// TIA Portal project "Automação_Grupo_2_V0.2" (V16)

(* hardware
DEVICE "S7-1200 station_1"  S7-1200 Station
   slot 0: "Rack_0"  S7-1200 Rack  Rack  V1.0
   slot 1: "PLC_1"  CPU 1211C AC/DC/Rly  6ES7 211-1BE40-0XB0  V4.4
   slot 3: "DI 4x24VDC_1"  DI4 signal board (200 kHz)  6ES7 221-3BD30-0XB0  V1.0
*)

// ===== PLC "PLC_1"  CPU 1211C AC/DC/Rly =====

VAR_GLOBAL   // PLC tag table "Default tag table"
   "Start(NO)" AT %I0.0 : Bool;
   "Stop(NC)" AT %I0.1 : Bool;
   "Reset(NO)" AT %I0.2 : Bool;
   "Emergência(NO)" AT %I0.3 : Bool;
   "Sensor Final (NO) AV PART1" AT %I0.4 : Bool;
   "Cilindro Alimentador Avanço" AT %I0.5 : Bool;
   "Peça no Alimentador" AT %I1.0 : Bool;
   "Sensor Fase 1 (NO)" AT %I1.1 : Bool;
   "Sensor Fase 2 (NO)" AT %I1.2 : Bool;
   "Sensor Fase 3 (NC)" AT %I1.3 : Bool;
   "Ordem Direita" AT %Q0.0 : Bool;
   "Ordem Esquerda" AT %Q0.1 : Bool;
   "Avanço Cilindro de Alimentação" AT %Q0.2 : Bool;
   "Seletor de Peças do Conveyor" AT %Q0.3 : Bool;
   "E_Verificação" AT %M0.1 : Bool;
   "E_2" AT %M0.2 : Bool;
   "E_3" AT %M0.3 : Bool;
   "E_4" AT %M0.4 : Bool;
   "E_5" AT %M0.5 : Bool;
   "E_6" AT %M0.6 : Bool;
   "E_7" AT %M0.7 : Bool;
   "E_8" AT %M1.0 : Bool;
   "E_9" AT %M1.1 : Bool;
   "E_10" AT %M1.2 : Bool;
   "T1_STATUS" AT %M1.3 : Bool;
END_VAR

// folder: System blocks/Program resources

DATA_BLOCK "T1"   // DB1
{ S7_Optimized_Access := 'TRUE' }
AUTHOR : Simatic
FAMILY : IEC
NAME : IEC_TMR
VERSION : 1.0
// stored: InstanceOfName IEC_TIMER
"IEC_TIMER"
BEGIN
END_DATA_BLOCK

DATA_BLOCK "Temporizador 01"   // DB2
{ S7_Optimized_Access := 'TRUE' }
AUTHOR : Simatic
FAMILY : IEC
NAME : IEC_TMR
VERSION : 1.0
// stored: InstanceOfName IEC_TIMER
"IEC_TIMER"
BEGIN
END_DATA_BLOCK

DATA_BLOCK "Cooldown para Motor"   // DB3
{ S7_Optimized_Access := 'TRUE' }
AUTHOR : Simatic
FAMILY : IEC
NAME : IEC_TMR
VERSION : 1.0
// stored: InstanceOfName IEC_TIMER
"IEC_TIMER"
BEGIN
END_DATA_BLOCK

DATA_BLOCK "COoldown para Desligar Esquerda"   // DB4
{ S7_Optimized_Access := 'TRUE' }
AUTHOR : Simatic
FAMILY : IEC
NAME : IEC_TMR
VERSION : 1.0
// stored: InstanceOfName IEC_TIMER
"IEC_TIMER"
BEGIN
END_DATA_BLOCK

DATA_BLOCK "Temporizador para Direita"   // DB5
{ S7_Optimized_Access := 'TRUE' }
AUTHOR : Simatic
FAMILY : IEC
NAME : IEC_TMR
VERSION : 1.0
// stored: InstanceOfName IEC_TIMER
"IEC_TIMER"
BEGIN
END_DATA_BLOCK

DATA_BLOCK "XTempo do Seletor"   // DB6
{ S7_Optimized_Access := 'TRUE' }
AUTHOR : Simatic
FAMILY : IEC
NAME : IEC_TMR
VERSION : 1.0
// stored: InstanceOfName IEC_TIMER
"IEC_TIMER"
BEGIN
END_DATA_BLOCK

DATA_BLOCK "Cooldown Estação 2"   // DB7
{ S7_Optimized_Access := 'TRUE' }
AUTHOR : Simatic
FAMILY : IEC
NAME : IEC_TMR
VERSION : 1.0
// stored: InstanceOfName IEC_TIMER
"IEC_TIMER"
BEGIN
END_DATA_BLOCK

DATA_BLOCK "5 Segundos 2a Estação"   // DB8
{ S7_Optimized_Access := 'TRUE' }
AUTHOR : Simatic
FAMILY : IEC
NAME : IEC_TMR
VERSION : 1.0
// stored: InstanceOfName IEC_TIMER
"IEC_TIMER"
BEGIN
END_DATA_BLOCK

DATA_BLOCK "Cooldown para fechar o Seletor"   // DB9
{ S7_Optimized_Access := 'TRUE' }
AUTHOR : Simatic
FAMILY : IEC
NAME : IEC_TMR
VERSION : 1.0
// stored: InstanceOfName IEC_TIMER
"IEC_TIMER"
BEGIN
END_DATA_BLOCK

DATA_BLOCK "Cooldown para Terminar Processo"   // DB10
{ S7_Optimized_Access := 'TRUE' }
AUTHOR : Simatic
FAMILY : IEC
NAME : IEC_TMR
VERSION : 1.0
// stored: InstanceOfName IEC_TIMER
"IEC_TIMER"
BEGIN
END_DATA_BLOCK

DATA_BLOCK "Cooldown para DEsligar mOtor 3a Estação"   // DB11
{ S7_Optimized_Access := 'TRUE' }
AUTHOR : Simatic
FAMILY : IEC
NAME : IEC_TMR
VERSION : 1.0
// stored: InstanceOfName IEC_TIMER
"IEC_TIMER"
BEGIN
END_DATA_BLOCK

DATA_BLOCK "condição de entrada e8+e9"   // DB12
{ S7_Optimized_Access := 'TRUE' }
AUTHOR : Simatic
FAMILY : IEC
NAME : IEC_TMR
VERSION : 1.0
// stored: InstanceOfName IEC_TIMER
"IEC_TIMER"
BEGIN
END_DATA_BLOCK

DATA_BLOCK "contador de peças"   // DB13
{ S7_Optimized_Access := 'TRUE' }
AUTHOR : Simatic
FAMILY : IEC
NAME : CNTR
VERSION : 1.0
// stored: InstanceOfName IEC_COUNTER
"IEC_COUNTER"
BEGIN
END_DATA_BLOCK

DATA_BLOCK "cooldown para mandar pecas novamente"   // DB14
{ S7_Optimized_Access := 'TRUE' }
AUTHOR : Simatic
FAMILY : IEC
NAME : IEC_TMR
VERSION : 1.0
// stored: InstanceOfName IEC_TIMER
"IEC_TIMER"
BEGIN
END_DATA_BLOCK

DATA_BLOCK "cooldown final"   // DB15
{ S7_Optimized_Access := 'TRUE' }
AUTHOR : Simatic
FAMILY : IEC
NAME : IEC_TMR
VERSION : 1.0
// stored: InstanceOfName IEC_TIMER
"IEC_TIMER"
BEGIN
END_DATA_BLOCK

DATA_BLOCK "cooldown para peça retirada"   // DB16
{ S7_Optimized_Access := 'TRUE' }
AUTHOR : Simatic
FAMILY : IEC
NAME : IEC_TMR
VERSION : 1.0
// stored: InstanceOfName IEC_TIMER
"IEC_TIMER"
BEGIN
END_DATA_BLOCK

// folder: (top level)

FUNCTION "Geral" : Void   // FC1, LAD
{ S7_Optimized_Access := 'TRUE' }
VERSION : 0.1
BEGIN

REGION Network 1: Input Inicial
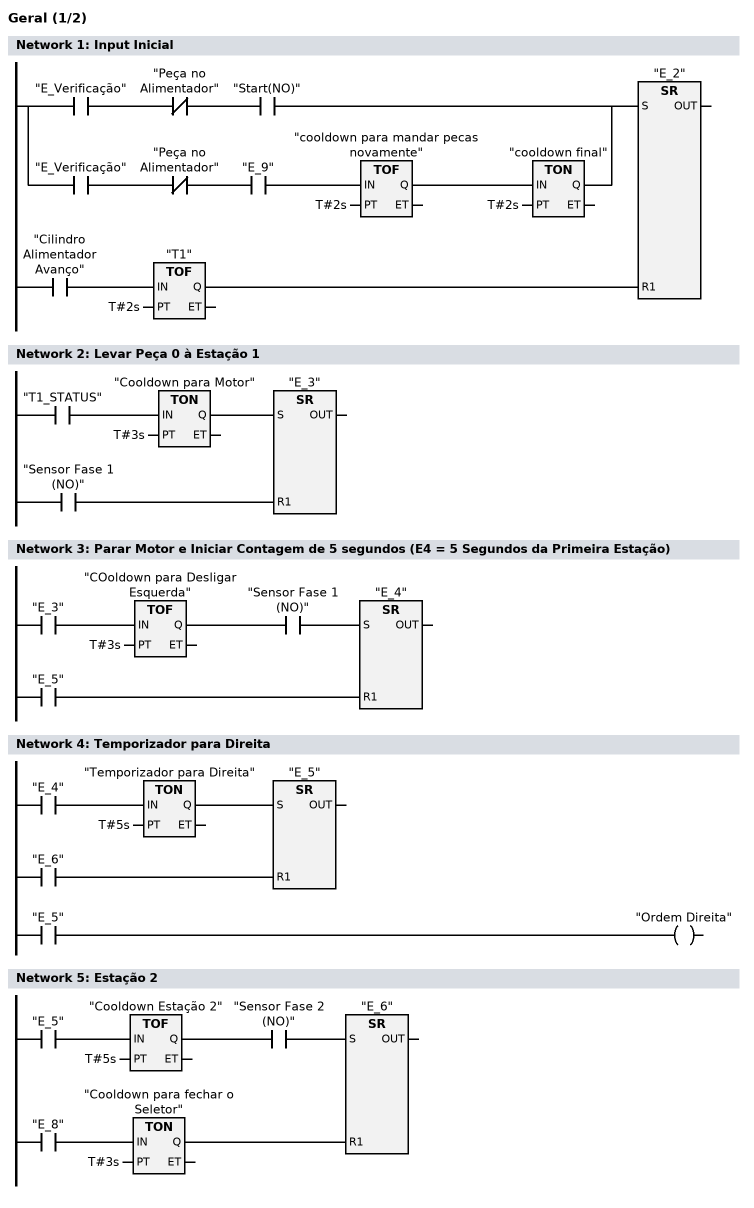
   "cooldown para mandar pecas novamente".TOF(IN := "E_Verificação" AND NOT "Peça no Alimentador" AND "E_9",
                           PT := T#2s);
   "cooldown final".TON(IN := "cooldown para mandar pecas novamente".Q, PT := T#2s);
   "T1".TOF(IN := "Cilindro Alimentador Avanço", PT := T#2s);
   IF ("E_Verificação" AND NOT "Peça no Alimentador" AND "Start(NO)") OR "cooldown final".Q THEN
       "E_2" := TRUE;   // SR flip-flop
   END_IF;
   IF "T1".Q THEN "E_2" := FALSE; END_IF;
END_REGION

REGION Network 2: Levar Peça 0 à Estação 1
   "Cooldown para Motor".TON(IN := "T1_STATUS", PT := T#3s);
   IF "Cooldown para Motor".Q THEN
       "E_3" := TRUE;   // SR flip-flop
   END_IF;
   IF "Sensor Fase 1 (NO)" THEN "E_3" := FALSE; END_IF;
END_REGION

REGION Network 3: Parar Motor e Iniciar Contagem de 5 segundos (E4 = 5 Segundos da Primeira Estação)
   "COoldown para Desligar Esquerda".TOF(IN := "E_3", PT := T#3s);
   IF "COoldown para Desligar Esquerda".Q AND "Sensor Fase 1 (NO)" THEN
       "E_4" := TRUE;   // SR flip-flop
   END_IF;
   IF "E_5" THEN "E_4" := FALSE; END_IF;
END_REGION

REGION Network 4: Temporizador para Direita
   "Temporizador para Direita".TON(IN := "E_4", PT := T#5s);
   IF "Temporizador para Direita".Q THEN
       "E_5" := TRUE;   // SR flip-flop
   END_IF;
   IF "E_6" THEN "E_5" := FALSE; END_IF;
   "Ordem Direita" := "E_5";
END_REGION

REGION Network 5: Estação 2
   "Cooldown Estação 2".TOF(IN := "E_5", PT := T#5s);
   "Cooldown para fechar o Seletor".TON(IN := "E_8", PT := T#3s);
   IF "Cooldown Estação 2".Q AND "Sensor Fase 2 (NO)" THEN
       "E_6" := TRUE;   // SR flip-flop
   END_IF;
   IF "Cooldown para fechar o Seletor".Q THEN "E_6" := FALSE; END_IF;
END_REGION

REGION Network 6: Controle de Ordens 2a Estação
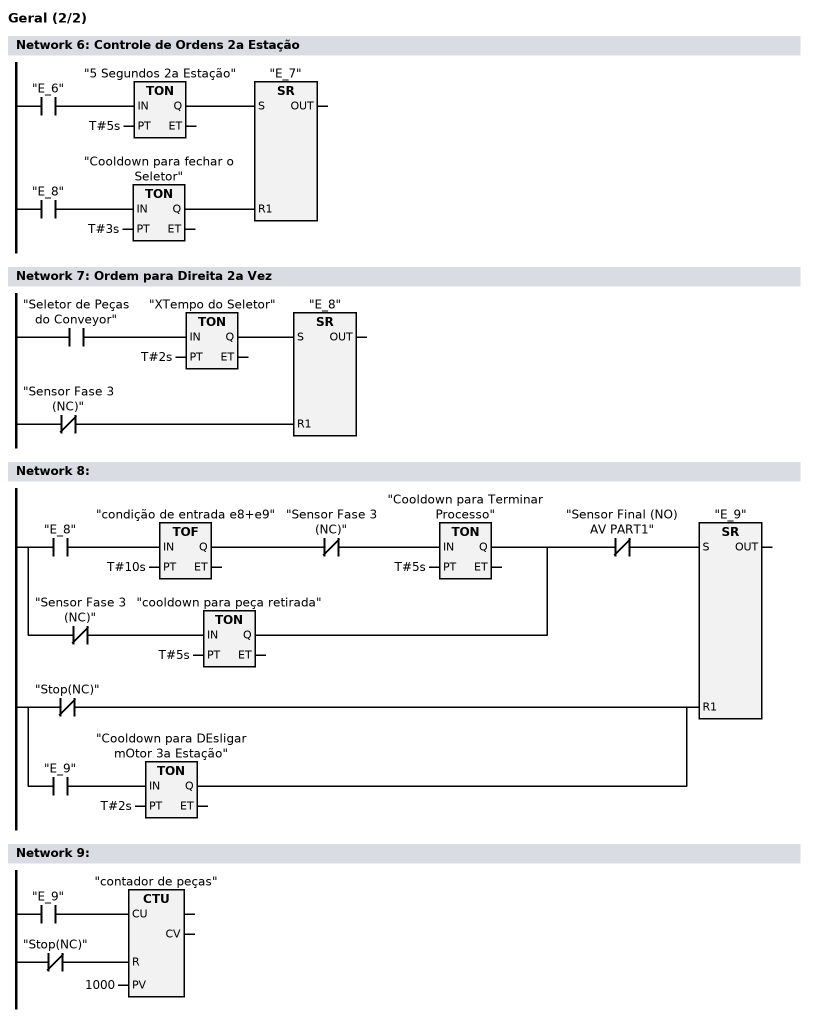
   "5 Segundos 2a Estação".TON(IN := "E_6", PT := T#5s);
   "Cooldown para fechar o Seletor".TON(IN := "E_8", PT := T#3s);
   IF "5 Segundos 2a Estação".Q THEN
       "E_7" := TRUE;   // SR flip-flop
   END_IF;
   IF "Cooldown para fechar o Seletor".Q THEN "E_7" := FALSE; END_IF;
END_REGION

REGION Network 7: Ordem para Direita 2a Vez
   "XTempo do Seletor".TON(IN := "Seletor de Peças do Conveyor", PT := T#2s);
   IF "XTempo do Seletor".Q THEN
       "E_8" := TRUE;   // SR flip-flop
   END_IF;
   IF NOT "Sensor Fase 3 (NC)" THEN "E_8" := FALSE; END_IF;
END_REGION

REGION Network 8
   "condição de entrada e8+e9".TOF(IN := "E_8", PT := T#10s);
   "Cooldown para Terminar Processo".TON(IN := "condição de entrada e8+e9".Q AND NOT "Sensor Fase 3 (NC)",
                           PT := T#5s);
   "cooldown para peça retirada".TON(IN := NOT "Sensor Fase 3 (NC)", PT := T#5s);
   "Cooldown para DEsligar mOtor 3a Estação".TON(IN := "E_9", PT := T#2s);
   IF ("Cooldown para Terminar Processo".Q OR "cooldown para peça retirada".Q) AND NOT "Sensor Final (NO) AV PART1" THEN
       "E_9" := TRUE;   // SR flip-flop
   END_IF;
   IF NOT "Stop(NC)" OR "Cooldown para DEsligar mOtor 3a Estação".Q THEN "E_9" := FALSE; END_IF;
END_REGION

REGION Network 9
   "contador de peças".CTU(CU := "E_9", R := NOT "Stop(NC)", PV := 1000);
END_REGION
END_FUNCTION

FUNCTION "Outputs" : Void   // FC2, LAD
{ S7_Optimized_Access := 'TRUE' }
VERSION : 0.1
BEGIN

REGION Network 1: Avanço Cilindro
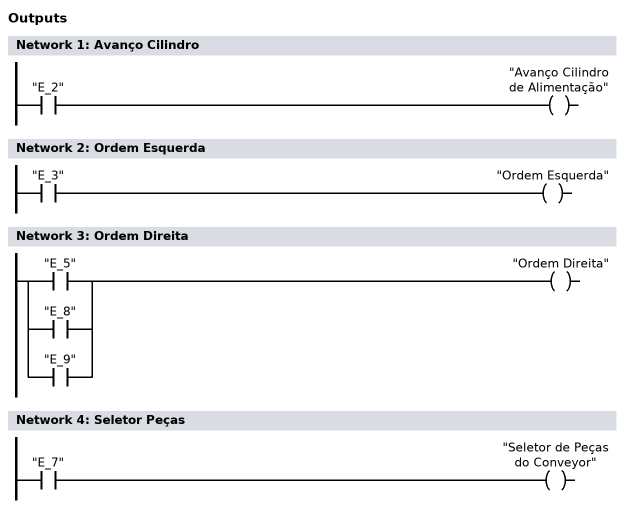
   RUNG wire#powerrail
      Contact( "E_2" )
      Coil( "Avanço Cilindro de Alimentação" )
   END_RUNG
   // the same network as SCL:
   "Avanço Cilindro de Alimentação" := "E_2";
END_REGION

REGION Network 2: Ordem Esquerda
   RUNG wire#powerrail
      Contact( "E_3" )
      Coil( "Ordem Esquerda" )
   END_RUNG
   // the same network as SCL:
   "Ordem Esquerda" := "E_3";
END_REGION

REGION Network 3: Ordem Direita
   RUNG wire#powerrail
      Contact( "E_5" )
      wire#w1
      Coil( "Ordem Direita" )
   END_RUNG
   RUNG wire#powerrail
      Contact( "E_8" )
   END_RUNG wire#w1
   RUNG wire#powerrail
      Contact( "E_9" )
   END_RUNG wire#w1
   // the same network as SCL:
   "Ordem Direita" := "E_5" OR "E_8" OR "E_9";
END_REGION

REGION Network 4: Seletor Peças
   RUNG wire#powerrail
      Contact( "E_7" )
      Coil( "Seletor de Peças do Conveyor" )
   END_RUNG
   // the same network as SCL:
   "Seletor de Peças do Conveyor" := "E_7";
END_REGION
END_FUNCTION

FUNCTION "Timers" : Void   // FC3, LAD
{ S7_Optimized_Access := 'TRUE' }
VERSION : 0.1
BEGIN

REGION Network 1: T1_Status
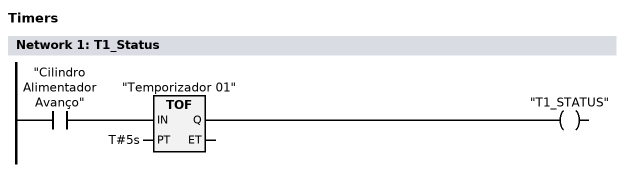
   "Temporizador 01".TOF(IN := "Cilindro Alimentador Avanço", PT := T#5s);
   "T1_STATUS" := "Temporizador 01".Q;
END_REGION
END_FUNCTION

FUNCTION "Sensors_Verification" : Void   // FC4, LAD
{ S7_Optimized_Access := 'TRUE' }
VERSION : 0.1
BEGIN

REGION Network 1: Verificação de Sensores
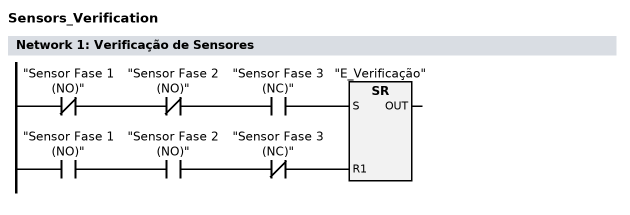
   RUNG wire#powerrail
      I_Contact( "Sensor Fase 1 (NO)" )
      I_Contact( "Sensor Fase 2 (NO)" )
      Contact( "Sensor Fase 3 (NC)" )
      S_SR(operand := "E_Verificação", r1 := wire#w1)
   END_RUNG
   RUNG wire#powerrail
      Contact( "Sensor Fase 1 (NO)" )
      Contact( "Sensor Fase 2 (NO)" )
      I_Contact( "Sensor Fase 3 (NC)" )
   END_RUNG wire#w1
   // the same network as SCL:
   IF NOT "Sensor Fase 1 (NO)" AND NOT "Sensor Fase 2 (NO)" AND "Sensor Fase 3 (NC)" THEN
       "E_Verificação" := TRUE;   // SR flip-flop
   END_IF;
   IF "Sensor Fase 1 (NO)" AND "Sensor Fase 2 (NO)" AND NOT "Sensor Fase 3 (NC)" THEN
       "E_Verificação" := FALSE;
   END_IF;
END_REGION
END_FUNCTION

ORGANIZATION_BLOCK "Main"   // OB1, LAD, ProgramCycle
TITLE = "Main Program Sweep (Cycle)"
{ S7_Optimized_Access := 'TRUE' }
VERSION : 0.1
   VAR_INPUT
      Initial_Call : Bool;   // Initial call of this OB
      Remanence : Bool;   // =True, if remanent data are available
   END_VAR
BEGIN

REGION Network 1
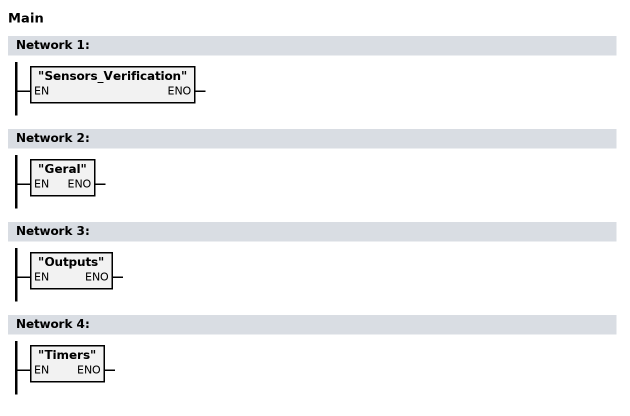
   RUNG wire#powerrail
      "Sensors_Verification"()
   END_RUNG
   // the same network as SCL:
   "Sensors_Verification"();
END_REGION

REGION Network 2
   RUNG wire#powerrail
      "Geral"()
   END_RUNG
   // the same network as SCL:
   "Geral"();
END_REGION

REGION Network 3
   RUNG wire#powerrail
      "Outputs"()
   END_RUNG
   // the same network as SCL:
   "Outputs"();
END_REGION

REGION Network 4
   RUNG wire#powerrail
      "Timers"()
   END_RUNG
   // the same network as SCL:
   "Timers"();
END_REGION
END_ORGANIZATION_BLOCK